// TIA Portal V17 export
// export: Created 2025-03-10T13:12:00.419977Z, ExportSetting WithDefaults, DisplayName Totally Integrated Automation Portal, DisplayVersion V17 Update 8, DisplayName TIA Portal Openness, DisplayVersion V17 Update 8, DisplayName TIA Portal Version Control Interface, DisplayVersion V17, DisplayName SINAMICS Startdrive Advanced, DisplayVersion V17 SP2, DisplayName SINAMICS Startdrive G110M, G120, G120C, G120D, G120P, G115D, DisplayVersion V17 SP2, DisplayName SINAMICS Startdrive G130, G150, S120, S150, SINAMICS MV, S210, DisplayVersion V17 SP2, DisplayName STEP 7 Professional, DisplayVersion V17 Update 8, DisplayName SINUMERIK ONE STEP 7 Toolbox, DisplayVersion V17 Update 12, DisplayName SINUMERIK 840D sl STEP 7 Toolbox, DisplayVersion V17 Update 12, DisplayName STEP 7 Safety, DisplayVersion V17 Update 6, DisplayName WinCC Advanced, DisplayVersion V17 Update 8
TYPE "LBP_typeModularMcpKeypadRecord"
TITLE = Modular MCP image / Imagen de MCP modulares / Abbild modulare MCP
// Image of modular MCP for key properties / Imagen de los MCP modulares para propiedades de las teclas / Abbild der modularen MCP für Tasteneigenschaften
// stored: IsFailsafeCompliant false
   STRUCT
      recordVersion : Byte := 16#10;   // Version 1.0 / version 1.0 / Versión 1.0
      keyActiveAttributesCount : USInt;   // Anzahl gültige Einträge in keyActiveAttributes / number of valid entries in keyActiveAttributes / Número de entradas válidas en keyActiveAttributes
      keyInactiveAttributesCount : USInt;   // Anzahl gültige Einträge in keyInactiveAttributes / number of valid entries in keyInactiveAttributes / Número de entradas válidas en keyInactiveAttributes
      reserved : Byte;   // Nicht verwendete Variable / unused variable / Variable no utilizada
      keyActiveAttributes { S7_SetPoint := 'True'} : Array[0..20] of "LBP_typeModularMcpLedAttribute";   // Farbattribute für Tasten im Status "active" / color attributes for keys in state "active" / Atributos de color para teclas en estado "activo"
      keyInactiveAttributes { S7_SetPoint := 'True'} : Array[0..20] of "LBP_typeModularMcpLedAttribute";   // Farbattribute für Tasten im Status "inactive" / color attributes for keys in state "inactive" / Atributos de color para teclas en estado "inactivo"
   END_STRUCT;
END_TYPE
